{attribute 'pack_mode' := '2'}
TYPE ST_CAM_INFO :
STRUCT
  bError              : BIT;
  wCamCouplingState   : ARRAY[0..7] OF WORD;
  nCamCouplingTableId : ARRAY[0..7] OF UINT;

  nNumPointsRead      : UDINT;
END_STRUCT
END_TYPE

(* stored: Version 1.1.0.1, ProductVersion 3.1.4024.12
   DUT ST_CAM_INFO: Id {071665c8-af33-0eb5-0770-2e8f064bb1fc} *)
